// TIA Portal V15.1 export
// export: Created 2025-12-09T12:24:19.1795411Z, ExportSetting WithDefaults, WithReadOnly, DisplayName Totally Integrated Automation Portal, DisplayVersion V15.1, DisplayName TIA Portal Openness, DisplayVersion V15.1, DisplayName SINAMICS Startdrive Advanced, DisplayVersion V15.1, DisplayName SINAMICS DCC, DisplayVersion V15.1, DisplayName G130, G150, S120, S150, SINAMICS MV, S210, DisplayVersion V15.1, DisplayName G110M, G120, G120C, G120D, G120P, DisplayVersion V15.1, DisplayName STEP 7 Professional, DisplayVersion V15.1, DisplayName STEP 7 Safety, DisplayVersion V15.1, DisplayName WinCC Professional, DisplayVersion V15.1, DisplayName SIMATIC Visualization Architect, DisplayVersion V15.1
DATA_BLOCK "[nome_robo][nome_ferramenta]#FB_Rob_Kleben_DB"   // DB[numero_db]
{ S7_Optimized_Access := 'TRUE'; DB_Accessible_From_OPC_UA := 'FALSE' }
AUTHOR : VASS_V06
FAMILY : ROBKL
NAME : ROBKL
VERSION : 0.1
// Kleben
// stored: AutoNumber false, CodeModifiedDate 2019-03-26T12:23:48.8112847Z, CompileDate 2019-04-01T14:36:08.7515261Z, CreationDate 2018-09-21T13:35:06.9687212Z, DBAccessibleFromOPCUA false, DownloadWithoutReinit false, InstanceOfName FB_Rob_Kleben, InstanceOfNumber 252, InstanceOfType FB, InterfaceModifiedDate 2019-03-01T11:50:30.6337089Z, IsConsistent true, IsKnowHowProtected false, IsRetainMemResEnabled false, MemoryReserve 0, ModifiedDate 2019-03-26T12:23:48.8112847Z, ParameterModified 2018-08-24T12:46:03.7885498Z, StructureModified 2018-09-22T16:29:23.4358261Z, UDAEnableTagReadback false
"FB_Rob_Kleben"
   // VAR_INPUT
   //    FrgAnwahl { ExternalAccessible := 'False'; ExternalVisible := 'False'; ExternalWritable := 'False'} : Bool;
   //    Option { ExternalAccessible := 'False'; ExternalVisible := 'False'; ExternalWritable := 'False'} : Int;
   //    Layer { ExternalAccessible := 'False'; ExternalVisible := 'False'; ExternalWritable := 'False'} : Int;
   //    Ex_Anwahl { ExternalAccessible := 'False'; ExternalVisible := 'False'; ExternalWritable := 'False'} : Word;
   //    Cfg { ExternalAccessible := 'False'; ExternalVisible := 'False'; ExternalWritable := 'False'} : Word;
   //    BMK_NR { ExternalAccessible := 'False'; ExternalVisible := 'False'; ExternalWritable := 'False'} : Byte;
   //    VkStoe_In { ExternalAccessible := 'False'; ExternalVisible := 'False'; ExternalWritable := 'False'} : Bool;
   // END_VAR
   // VAR_OUTPUT
   //    ohneProz { ExternalAccessible := 'False'; ExternalVisible := 'False'; ExternalWritable := 'False'} : Bool;
   //    PA { ExternalAccessible := 'False'; ExternalVisible := 'False'; ExternalWritable := 'False'} : Bool;
   //    Ex_LM { ExternalAccessible := 'False'; ExternalVisible := 'False'; ExternalWritable := 'False'} : Word;
   //    Vorw { ExternalAccessible := 'False'; ExternalVisible := 'False'; ExternalWritable := 'False'} : Bool;
   //    Stoexx { ExternalAccessible := 'False'; ExternalVisible := 'False'; ExternalWritable := 'False'} : Bool;
   //    Vk_Stoe_Out { ExternalAccessible := 'False'; ExternalVisible := 'False'; ExternalWritable := 'False'} : Bool;
   // END_VAR
   // VAR_IN_OUT
   //    ST_ROB : "ST_Rob";
   //    ST_PG : "ST_PG";
   //    ST_BA : "ST_Betriebsarten";
   // END_VAR
   // VAR RETAIN
   //    "HMI-UDT" : "HMI-UDT_Rob_Kleben";
   // END_VAR
   // VAR
   //    "001" { ExternalAccessible := 'False'; ExternalVisible := 'False'; ExternalWritable := 'False'} : Bool;
   //    "002" { ExternalAccessible := 'False'; ExternalVisible := 'False'; ExternalWritable := 'False'} : Bool;
   //    "003" { ExternalAccessible := 'False'; ExternalVisible := 'False'; ExternalWritable := 'False'} : Bool;
   //    "004" { ExternalAccessible := 'False'; ExternalVisible := 'False'; ExternalWritable := 'False'} : Bool;
   //    "005" { ExternalAccessible := 'False'; ExternalVisible := 'False'; ExternalWritable := 'False'} : Bool;
   //    "006" { ExternalAccessible := 'False'; ExternalVisible := 'False'; ExternalWritable := 'False'} : Bool;
   //    "007" { ExternalAccessible := 'False'; ExternalVisible := 'False'; ExternalWritable := 'False'} : Bool;
   //    "008" { ExternalAccessible := 'False'; ExternalVisible := 'False'; ExternalWritable := 'False'} : Bool;
   //    "009" { ExternalAccessible := 'False'; ExternalVisible := 'False'; ExternalWritable := 'False'} : Bool;
   //    "010" { ExternalAccessible := 'False'; ExternalVisible := 'False'; ExternalWritable := 'False'} : Bool;
   //    "011" { ExternalAccessible := 'False'; ExternalVisible := 'False'; ExternalWritable := 'False'} : Bool;
   //    "012" { ExternalAccessible := 'False'; ExternalVisible := 'False'; ExternalWritable := 'False'} : Bool;
   //    "013" { ExternalAccessible := 'False'; ExternalVisible := 'False'; ExternalWritable := 'False'} : Bool;
   //    "014" { ExternalAccessible := 'False'; ExternalVisible := 'False'; ExternalWritable := 'False'} : Bool;
   //    "015" { ExternalAccessible := 'False'; ExternalVisible := 'False'; ExternalWritable := 'False'} : Bool;
   //    "255" { ExternalAccessible := 'False'; ExternalVisible := 'False'; ExternalWritable := 'False'} : Bool;
   // END_VAR
   // VAR RETAIN
   //    ST_GlobAnwProz { ExternalAccessible := 'False'; ExternalVisible := 'False'; ExternalWritable := 'False'} : "HMI-UDT_GlobAnw";
   // END_VAR
   // VAR
   //    xSF_oProz { ExternalAccessible := 'False'; ExternalVisible := 'False'; ExternalWritable := 'False'} : Bool;
   //    xSF_Pistole1 { ExternalAccessible := 'False'; ExternalVisible := 'False'; ExternalWritable := 'False'} : Bool;
   //    xSF_Pistole2 { ExternalAccessible := 'False'; ExternalVisible := 'False'; ExternalWritable := 'False'} : Bool;
   //    xSF_Zeigen { ExternalAccessible := 'False'; ExternalVisible := 'False'; ExternalWritable := 'False'} : Bool;
   //    xSF_Spuelen { ExternalAccessible := 'False'; ExternalVisible := 'False'; ExternalWritable := 'False'} : Bool;
   //    xSF_BTiO { ExternalAccessible := 'False'; ExternalVisible := 'False'; ExternalWritable := 'False'} : Bool;
   //    xSF_BTAuss { ExternalAccessible := 'False'; ExternalVisible := 'False'; ExternalWritable := 'False'} : Bool;
   //    xSF_BTNaArb { ExternalAccessible := 'False'; ExternalVisible := 'False'; ExternalWritable := 'False'} : Bool;
   //    xSF_Wart { ExternalAccessible := 'False'; ExternalVisible := 'False'; ExternalWritable := 'False'} : Bool;
   //    xSF_HzNt { ExternalAccessible := 'False'; ExternalVisible := 'False'; ExternalWritable := 'False'} : Bool;
   //    xSF_HzAus { ExternalAccessible := 'False'; ExternalVisible := 'False'; ExternalWritable := 'False'} : Bool;
   // END_VAR
   // VAR RETAIN
   //    xGlobSk_oProz { ExternalAccessible := 'False'; ExternalVisible := 'False'; ExternalWritable := 'False'} : Bool;
   //    xGlobSk_Pistole1 { ExternalAccessible := 'False'; ExternalVisible := 'False'; ExternalWritable := 'False'} : Bool;
   //    xGlobSk_Pistole2 { ExternalAccessible := 'False'; ExternalVisible := 'False'; ExternalWritable := 'False'} : Bool;
   //    xGlobSk_Wartung { ExternalAccessible := 'False'; ExternalVisible := 'False'; ExternalWritable := 'False'} : Bool;
   //    xAnwPistole1 { ExternalAccessible := 'False'; ExternalVisible := 'False'; ExternalWritable := 'False'} : Bool;
   //    xAnwPistole2 { ExternalAccessible := 'False'; ExternalVisible := 'False'; ExternalWritable := 'False'} : Bool;
   //    xAnwPistole3 { ExternalAccessible := 'False'; ExternalVisible := 'False'; ExternalWritable := 'False'} : Bool;
   //    xAnwZeigen { ExternalAccessible := 'False'; ExternalVisible := 'False'; ExternalWritable := 'False'} : Bool;
   //    xAnwSpuelen { ExternalAccessible := 'False'; ExternalVisible := 'False'; ExternalWritable := 'False'} : Bool;
   //    xWartung_Spuelen { ExternalAccessible := 'False'; ExternalVisible := 'False'; ExternalWritable := 'False'} : Bool;
   //    strOption_Alt { ExternalAccessible := 'False'; ExternalVisible := 'False'; ExternalWritable := 'False'} : Int;
   // END_VAR
   // VAR
   //    xZG_Rueckmeldung { ExternalAccessible := 'False'; ExternalVisible := 'False'; ExternalWritable := 'False'} : Bool;
   //    xSP_Rueckmeldung { ExternalAccessible := 'False'; ExternalVisible := 'False'; ExternalWritable := 'False'} : Bool;
   // END_VAR
   // VAR RETAIN
   //    xResetFlanke { ExternalAccessible := 'False'; ExternalVisible := 'False'; ExternalWritable := 'False'} : Bool;
   //    xQuit_BTiO { ExternalAccessible := 'False'; ExternalVisible := 'False'; ExternalWritable := 'False'} : Bool;
   //    xQuit_BTAuss { ExternalAccessible := 'False'; ExternalVisible := 'False'; ExternalWritable := 'False'} : Bool;
   //    xQuit_BTNaArb { ExternalAccessible := 'False'; ExternalVisible := 'False'; ExternalWritable := 'False'} : Bool;
   //    xQuit_B { ExternalAccessible := 'False'; ExternalVisible := 'False'; ExternalWritable := 'False'} : Bool;
   //    xEMode_Aus { ExternalAccessible := 'False'; ExternalVisible := 'False'; ExternalWritable := 'False'} : Bool;
   //    xEMode_Ein { ExternalAccessible := 'False'; ExternalVisible := 'False'; ExternalWritable := 'False'} : Bool;
   //    xHzAus { ExternalAccessible := 'False'; ExternalVisible := 'False'; ExternalWritable := 'False'} : Bool;
   //    bPrio { ExternalAccessible := 'False'; ExternalVisible := 'False'; ExternalWritable := 'False'} : Byte;
   //    iLayerIntern { ExternalAccessible := 'False'; ExternalVisible := 'False'; ExternalWritable := 'False'} : Int;
   // END_VAR
   // VAR
   //    xLayerNIO { ExternalAccessible := 'False'; ExternalVisible := 'False'; ExternalWritable := 'False'} : Bool;
   //    xLayerAktiv { ExternalAccessible := 'False'; ExternalVisible := 'False'; ExternalWritable := 'False'} : Bool;
   // END_VAR
   // VAR RETAIN
   //    xA_Len { ExternalAccessible := 'False'; ExternalVisible := 'False'; ExternalWritable := 'False'} : Bool;
   //    xOpt_Error1 { ExternalAccessible := 'False'; ExternalVisible := 'False'; ExternalWritable := 'False'} : Bool;
   //    xOpt_Error2 { ExternalAccessible := 'False'; ExternalVisible := 'False'; ExternalWritable := 'False'} : Bool;
   //    xOpt_Error3 { ExternalAccessible := 'False'; ExternalVisible := 'False'; ExternalWritable := 'False'} : Bool;
   //    iK_Adress1 { ExternalAccessible := 'False'; ExternalVisible := 'False'; ExternalWritable := 'False'} : Int;
   //    iK_Adress2 { ExternalAccessible := 'False'; ExternalVisible := 'False'; ExternalWritable := 'False'} : Int;
   //    iEA_Adress { ExternalAccessible := 'False'; ExternalVisible := 'False'; ExternalWritable := 'False'} : Int;
   //    strK { ExternalAccessible := 'False'; ExternalVisible := 'False'; ExternalWritable := 'False'} : String[25];
   //    PEiW { ExternalAccessible := 'False'; ExternalVisible := 'False'; ExternalWritable := 'False'} : Int;
   // END_VAR
   // VAR
   //    xVorw_Fass { ExternalAccessible := 'False'; ExternalVisible := 'False'; ExternalWritable := 'False'} : Bool;
   //    xVorw_la { ExternalAccessible := 'False'; ExternalVisible := 'False'; ExternalWritable := 'False'} : Bool;
   //    xEngspM_Ein { ExternalAccessible := 'False'; ExternalVisible := 'False'; ExternalWritable := 'False'} : Bool;
   //    xF_HPD { ExternalAccessible := 'False'; ExternalVisible := 'False'; ExternalWritable := 'False'} : Bool;
   //    xF_Kl { ExternalAccessible := 'False'; ExternalVisible := 'False'; ExternalWritable := 'False'} : Bool;
   //    xF_BB { ExternalAccessible := 'False'; ExternalVisible := 'False'; ExternalWritable := 'False'} : Bool;
   //    xStoe { ExternalAccessible := 'False'; ExternalVisible := 'False'; ExternalWritable := 'False'} : Bool;
   //    xF_PTemp { ExternalAccessible := 'False'; ExternalVisible := 'False'; ExternalWritable := 'False'} : Bool;
   // END_VAR
   // VAR RETAIN
   //    X_KL { ExternalAccessible := 'False'; ExternalVisible := 'False'; ExternalWritable := 'False'} : Byte;
   //    xSperre_Quit_BTNaArb { ExternalAccessible := 'False'; ExternalVisible := 'False'; ExternalWritable := 'False'} : Bool;
   //    xSG_Auf_Zu { ExternalAccessible := 'False'; ExternalVisible := 'False'; ExternalWritable := 'False'} : Bool;
   //    xSG_Auf_Zu_1 { ExternalAccessible := 'False'; ExternalVisible := 'False'; ExternalWritable := 'False'} : Bool;
   // END_VAR
   // VAR
   //    xInit { ExternalAccessible := 'False'; ExternalVisible := 'False'; ExternalWritable := 'False'} : Bool;
   // END_VAR
   // VAR RETAIN
   //    xStoexx { ExternalAccessible := 'False'; ExternalVisible := 'False'; ExternalWritable := 'False'} : Bool;
   //    xOhneProz { ExternalAccessible := 'False'; ExternalVisible := 'False'; ExternalWritable := 'False'} : Bool;
   // END_VAR
   // VAR
   //    R_TRIG_oProzGlobSk { ExternalAccessible := 'False'; ExternalVisible := 'False'; ExternalWritable := 'False'} : "R_Trig";
   //    R_TRIG_Layer { ExternalAccessible := 'False'; ExternalVisible := 'False'; ExternalWritable := 'False'} : "R_Trig";
   //    R_TRIG_Pistole1GlobSk { ExternalAccessible := 'False'; ExternalVisible := 'False'; ExternalWritable := 'False'} : "R_Trig";
   //    R_TRIG_Pistole2GlobSk { ExternalAccessible := 'False'; ExternalVisible := 'False'; ExternalWritable := 'False'} : "R_Trig";
   //    R_TRIG_WartungGlobSk { ExternalAccessible := 'False'; ExternalVisible := 'False'; ExternalWritable := 'False'} : "R_Trig";
   //    R_TRIG_Zeigen { ExternalAccessible := 'False'; ExternalVisible := 'False'; ExternalWritable := 'False'} : "R_Trig";
   //    F_TRIG_Zeigen { ExternalAccessible := 'False'; ExternalVisible := 'False'; ExternalWritable := 'False'} : "F_Trig";
   //    F_TRIG_Wart_ang { ExternalAccessible := 'False'; ExternalVisible := 'False'; ExternalWritable := 'False'} : "F_Trig";
   //    F_TRIG_Stoe { ExternalAccessible := 'False'; ExternalVisible := 'False'; ExternalWritable := 'False'} : "F_Trig";
   //    R_TRIG_AnAb_Pistole1 { ExternalAccessible := 'False'; ExternalVisible := 'False'; ExternalWritable := 'False'} : "R_Trig";
   //    R_TRIG_AnAb_Pistole2 { ExternalAccessible := 'False'; ExternalVisible := 'False'; ExternalWritable := 'False'} : "R_Trig";
   //    R_TRIG_Anw_Wart { ExternalAccessible := 'False'; ExternalVisible := 'False'; ExternalWritable := 'False'} : "R_Trig";
   //    R_TRIG_ZG_Anwahl { ExternalAccessible := 'False'; ExternalVisible := 'False'; ExternalWritable := 'False'} : "R_Trig";
   //    R_TRIG_oProz { ExternalAccessible := 'False'; ExternalVisible := 'False'; ExternalWritable := 'False'} : "R_Trig";
   //    R_TRIG_Wser { ExternalAccessible := 'False'; ExternalVisible := 'False'; ExternalWritable := 'False'} : "R_Trig";
   //    R_TRIG_Taste_BTiO { ExternalAccessible := 'False'; ExternalVisible := 'False'; ExternalWritable := 'False'} : "R_Trig";
   //    R_TRIG_Taste_BTAuss { ExternalAccessible := 'False'; ExternalVisible := 'False'; ExternalWritable := 'False'} : "R_Trig";
   //    R_TRIG_Taste_BTNaArb { ExternalAccessible := 'False'; ExternalVisible := 'False'; ExternalWritable := 'False'} : "R_Trig";
   //    R_TRIG_Wartung_Spuelen { ExternalAccessible := 'False'; ExternalVisible := 'False'; ExternalWritable := 'False'} : "R_Trig";
   //    R_TRIG_xS_EngspM { ExternalAccessible := 'False'; ExternalVisible := 'False'; ExternalWritable := 'False'} : "R_Trig";
   //    R_TRIG_xS_HzNt { ExternalAccessible := 'False'; ExternalVisible := 'False'; ExternalWritable := 'False'} : "R_Trig";
   //    R_TRIG_EngspM_Ein { ExternalAccessible := 'False'; ExternalVisible := 'False'; ExternalWritable := 'False'} : "R_Trig";
   //    R_TRIG_EngspM_Aus { ExternalAccessible := 'False'; ExternalVisible := 'False'; ExternalWritable := 'False'} : "R_Trig";
   //    R_TRIG_Spuelen { ExternalAccessible := 'False'; ExternalVisible := 'False'; ExternalWritable := 'False'} : "R_Trig";
   //    R_TRIG_AnwAbwerfen { ExternalAccessible := 'False'; ExternalVisible := 'False'; ExternalWritable := 'False'} : "R_Trig";
   //    R_TRIG_xSF_HzAus { ExternalAccessible := 'False'; ExternalVisible := 'False'; ExternalWritable := 'False'} : "R_Trig";
   //    R_TRIG_HzAus { ExternalAccessible := 'False'; ExternalVisible := 'False'; ExternalWritable := 'False'} : "R_Trig";
   //    F_TRIG_Wartung_Spuelen { ExternalAccessible := 'False'; ExternalVisible := 'False'; ExternalWritable := 'False'} : "F_Trig";
   //    F_TRIG_Wser { ExternalAccessible := 'False'; ExternalVisible := 'False'; ExternalWritable := 'False'} : "F_Trig";
   //    F_TRIG_Spuelen { ExternalAccessible := 'False'; ExternalVisible := 'False'; ExternalWritable := 'False'} : "F_Trig";
   //    F_TRIG_Opt_Error { ExternalAccessible := 'False'; ExternalVisible := 'False'; ExternalWritable := 'False'} : "F_Trig";
   // END_VAR
   // VAR RETAIN
   //    TON_EngspM_Ein { ExternalAccessible := 'False'; ExternalVisible := 'False'; ExternalWritable := 'False'} : TON_TIME;
   //    TON_EngspM_Aus { ExternalAccessible := 'False'; ExternalVisible := 'False'; ExternalWritable := 'False'} : TON_TIME;
   //    TON_Quit_BTNaArb { ExternalAccessible := 'False'; ExternalVisible := 'False'; ExternalWritable := 'False'} : TON_TIME;
   //    TON_xAnwSpuelen { ExternalAccessible := 'False'; ExternalVisible := 'False'; ExternalWritable := 'False'} : TON_TIME;
   //    TON_HzAus { ExternalAccessible := 'False'; ExternalVisible := 'False'; ExternalWritable := 'False'} : TON_TIME;
   // END_VAR
   // VAR
   //    FB_Rob_Option_1 { ExternalAccessible := 'False'; ExternalVisible := 'False'; ExternalWritable := 'False'} : "FB_Rob_Option";
   // END_VAR
BEGIN
END_DATA_BLOCK
